FUNCTION_BLOCK SS1_SS2_ifb_RobotWithTimer (* Composite FB wrapping other FBs *)
  (* Standard: 61499-2 *)
  (* Version 1.0, 2024-08-30, DEVIASH *)
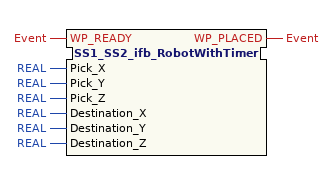
  EVENT_INPUT
    WP_READY; (* Initialization Request *)
  END_EVENT
  EVENT_OUTPUT
    WP_PLACED; (* Initialization Confirm *)
  END_EVENT
  VAR_INPUT
    Pick_X : REAL;
    Pick_Y : REAL;
    Pick_Z : REAL;
    Destination_X : REAL;
    Destination_Y : REAL;
    Destination_Z : REAL;
  END_VAR
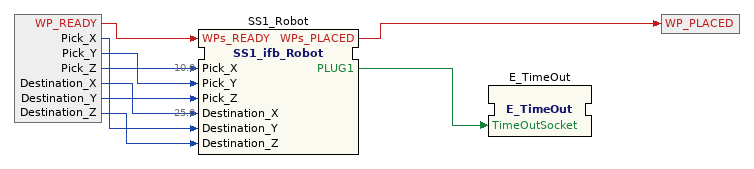
  FBS
    SS1_Robot : SS1_ifb_Robot(Pick_X := 10.0, Destination_X := 25.0);
    E_TimeOut : E_TimeOut;
  END_FBS
  EVENT_CONNECTIONS
    WP_READY TO SS1_Robot.WPs_READY;
    SS1_Robot.WPs_PLACED TO WP_PLACED;
  END_CONNECTIONS
  DATA_CONNECTIONS
    Pick_X TO SS1_Robot.Pick_X;
    Pick_Y TO SS1_Robot.Pick_Y;
    Pick_Z TO SS1_Robot.Pick_Z;
    Destination_X TO SS1_Robot.Destination_X;
    Destination_Y TO SS1_Robot.Destination_Y;
    Destination_Z TO SS1_Robot.Destination_Z;
  END_CONNECTIONS
  ADAPTER_CONNECTIONS
    SS1_Robot.PLUG1 TO E_TimeOut.TimeOutSocket;
  END_CONNECTIONS
END_FUNCTION_BLOCK
